(* PLC project Generated.project, CODESYS CODESYS V3.5 SP19 Patch 1 *)
(* stored: creationDateTime 2026-09-06T13:00:42.375521, modificationDateTime 2026-09-06T13:00:42.375521 *)

(* ======================================================================= 📊 ST_Diag_Device — Structure diagnostic d'un esclave ou bus ─────────────────────────────────────────────────────────────── 🎯 Rôle : Structure de donnees d'état, diagnostic et alarme d'un equipement réseau 📄 Doc métier : DOC/AF/AF_Partie-12_Fonction_Diagnostic_v1.4.md ======================================================================= *)
TYPE ST_Diag_Device : STRUCT
  Online : BOOL;  (* Esclave visible sur le bus *)
  Operational : BOOL;  (* Esclave en mode OP (opérationnel) *)
  Error : BOOL;  (* Signal de défaut actif pour cet esclave *)
  ErrorId : WORD;  (* Code défaut détaillé *)
  State : E_Diag_State;  (* Phase courante du cycle de diagnostic *)
  StateAtError : E_Diag_State;  (* Instantané de la phase lors de l'anomalie *)
END_STRUCT;
END_TYPE

(* values of E_Diag_State: DISABLED: Désactivé (surveillance non active); READY: Opérationnel réel, pas de défaut; INIT: Initialisation / Recherche de réseau; MONITORING: Surveillance active (états transitoires); ERROR: Anomalie de communication; SIMULATED: Bypass simulation ou bypass réseau IHM — pas le bus réel *)

{attribute 'qualified_only'}
{attribute 'strict'}
TYPE E_Diag_State : (DISABLED := 0, READY := 1, INIT := 2, MONITORING := 3, ERROR := 4, SIMULATED := 5);
END_TYPE
